INTERFACE I_ChunkedRequestSessionData EXTENDS I_SessionData

PROPERTY PUBLIC IsComplete : BOOL
GET
END_GET
END_PROPERTY

PROPERTY PUBLIC PayloadAddress : POINTER TO STRING
GET
END_GET
END_PROPERTY

PROPERTY PUBLIC PayloadSizeInBytes : UDINT
GET
END_GET
END_PROPERTY

METHOD PUBLIC TryAddChunkedPayload : BOOL;
VAR_INPUT
	PayloadAddress : POINTER TO STRING;
	PayloadSize : DINT;
	ChunkSequence : DINT;
END_VAR
END_METHOD

END_INTERFACE

(* stored: Version 1.1.0.1, ProductVersion 3.1.4024.12
   Itf I_ChunkedRequestSessionData: Id {22300d9d-d667-4bc8-b0b3-5a4fa8f36f5d}
   Property IsComplete: Id {dec49cc7-3ada-4338-bf34-8f28fd7fa0b6}
   Get Get: Id {f8c4caa5-5470-45d1-b7a7-46724b7937ce}
   Property PayloadAddress: Id {fe185271-e250-47aa-a0b9-2e0e28a991c8}
   Get Get: Id {8456e78e-25c8-4737-bab5-94ad02e875a7}
   Property PayloadSizeInBytes: Id {d690937c-d467-4628-a473-8fcf6c810e11}
   Get Get: Id {d5d17680-b9dc-4e35-b159-bc292786ec3f}
   Method TryAddChunkedPayload: Id {ea33a017-e809-4192-9e23-7f6dbb771687} *)
